FUNCTION_BLOCK FB_TCP_IP
VAR_INPUT
	sName				: STRING := 'SR1000';			(* A kódolvasó neve *)
	sRemoteHost			: STRING(15) := '127.0.0.1';	(* IP adress of remote server *)
	nRemotePort			: UDINT := 9004;				(* SR1000 default port *)
END_VAR
VAR_OUTPUT
END_VAR
VAR
	fbConnect 			:FB_SocketConnect;
	fbSend 				:FB_SocketSend;
	fbReceive 			:FB_SocketReceive;
	fbClose				:FB_SocketClose;
	sTxBuffer			:STRING;
	sRxBuffer			:STRING;
	nStep				:INT := 0;
	
	_ConnectTimeout		:TIME;
	_SendTimeout		:TIME;
	_ReceiveTimeout		:TIME;
	_CloseTimeout		:TIME;

END_VAR

(*
fbConnect(
	sSrvNetId:= '', 
	sRemoteHost:= sRemoteHost, 
	nRemotePort:= nRemotePort, 
	bExecute:= , 
	tTimeout:= _ConnectTimeout, 
	bBusy=> , 
	bError=> , 
	nErrId=> , 
	hSocket=> );
	
fbSend(
	sSrvNetId:= '', 
	hSocket:= fbConnect.hSocket, 
	cbLen:= INT_TO_UDINT(LEN(sTxBuffer)), 
	pSrc:= ADR(sTxBuffer), 
	bExecute:= , 
	tTimeout:= _SendTimeout, 
	bBusy=> , 
	bError=> , 
	nErrId=> );

fbReceive(
	sSrvNetId:= '', 
	hSocket:= fbConnect.hSocket, 
	cbLen:= SIZEOF(sRxBuffer), 
	pDest:= ADR(sRxBuffer), 
	bExecute:= , 
	tTimeout:= _ReceiveTimeout, 
	bBusy=> , 
	bError=> , 
	nErrId=> , 
	nRecBytes=> );

fbClose(
	sSrvNetId:= '', 
	hSocket:= fbConnect.hSocket, 
	bExecute:= , 
	tTimeout:= , 
	bBusy=> , 
	bError=> , 
	nErrId=> );	
	
*)

PROPERTY p_CloseTimeout :  TIME
GET
p_CloseTimeout := _CloseTimeout;
END_GET
SET
IF p_CloseTimeout > T#100MS AND p_CloseTimeout <  T#60S THEN
	_CloseTimeout := p_CloseTimeout;
ELSE
	_CloseTimeout := T#1S;					// default value
END_IF
END_SET
END_PROPERTY

PROPERTY p_ConnectTimeout : TIME
GET
p_ConnectTimeout := _ConnectTimeout;
END_GET
SET
IF p_ConnectTimeout > T#100MS AND p_ConnectTimeout <  T#60S THEN
	_ConnectTimeout := p_ConnectTimeout;
ELSE
	_ConnectTimeout := T#1S;					// default value
END_IF
END_SET
END_PROPERTY

PROPERTY p_ReceiveTimeout : TIME
GET
p_ReceiveTimeout := _ReceiveTimeout;
END_GET
SET
IF p_ReceiveTimeout > T#100MS AND p_ReceiveTimeout <  T#60S THEN
	_ReceiveTimeout := p_ReceiveTimeout;
ELSE
	_ReceiveTimeout := T#1S;					// default value
END_IF
END_SET
END_PROPERTY

PROPERTY p_SendTimeout : TIME
GET
p_SendTimeout := _SendTimeout;
END_GET
SET
IF p_SendTimeout > T#100MS AND p_SendTimeout <  T#60S THEN
	_SendTimeout := p_SendTimeout;
ELSE
	_SendTimeout := T#1S;					// default value
END_IF
END_SET
END_PROPERTY

METHOD ReadSR1000 : BOOL
VAR_INPUT
	sCode						:REFERENCE TO STRING;
	nErrorId					:REFERENCE TO UDINT;
END_VAR
TCP_Com();
ReadSR1000 := FALSE;
CASE nStep OF
0:		fbConnect.bExecute := TRUE;
		sRxBuffer := '';
		nStep := nStep + 20;
	
20:		IF NOT fbConnect.bBusy THEN
			fbConnect.bExecute := FALSE;
			nStep := nStep + 20;
		ELSIF fbConnect.bError THEN
			sCode := '';
			nErrorId := fbConnect.nErrId;
			fbConnect.bExecute := FALSE;
			nStep := 200;
		END_IF
	
40:		sTxBuffer := 'LON$R$N';
		fbSend.bExecute := TRUE;
		nStep := nStep + 20;
	
60:		IF NOT fbSend.bBusy THEN
			fbSend.bExecute := FALSE;
			nStep := 100;
		ELSIF fbSend.bError THEN
			sCode := '';
			nErrorId := fbSend.nErrId;
			fbSend.bExecute := FALSE;
			nStep := 200;
		END_IF
	
100:	fbReceive.bExecute := TRUE;
		nStep := nStep + 20;
	
120:	IF NOT fbReceive.bBusy THEN
			IF NOT fbReceive.bError THEN
					fbReceive.bExecute := FALSE;
					nStep := nStep + 20;
			ELSE
					sCode := '';
					nErrorId := fbReceive.nErrId;
					fbReceive.bExecute := FALSE;
					nStep := 200;
			END_IF
		END_IF

140:	IF fbReceive.nRecBytes > 0 THEN
				IF MID(sRxBuffer, 1, UDINT_TO_INT(fbReceive.nRecBytes)) = '$0D' THEN
					nErrorId := fbReceive.nErrId;
					sCode := LEFT(sRxBuffer, UDINT_TO_INT(fbReceive.nRecBytes)-1);
					nStep := 200;
				ELSE				
					nStep := 100;
				END_IF
		ELSE
				nStep := 100;
		END_IF
		
200:	fbClose.bExecute := TRUE;
		nStep := nStep + 20;
	
220:	IF NOT fbClose.bBusy THEN
			fbClose.bExecute := FALSE;
			nStep := 500;
		ELSIF fbClose.bError THEN
			sCode := '';
			nErrorId := fbClose.nErrId;
			fbClose.bExecute := FALSE;
			nStep := 500;
		END_IF

500:
		ReadSR1000 := TRUE;
		nStep := 0;
END_CASE
END_METHOD

METHOD PRIVATE TCP_Com : BOOL
VAR_INPUT
END_VAR
fbConnect(
	sSrvNetId:= '', 
	sRemoteHost:= sRemoteHost, 
	nRemotePort:= nRemotePort, 
	bExecute:= , 
	tTimeout:= _ConnectTimeout, 
	bBusy=> , 
	bError=> , 
	nErrId=> , 
	hSocket=> );
	
fbSend(
	sSrvNetId:= '', 
	hSocket:= fbConnect.hSocket, 
	cbLen:= INT_TO_UDINT(LEN(sTxBuffer)), 
	pSrc:= ADR(sTxBuffer), 
	bExecute:= , 
	tTimeout:= _SendTimeout, 
	bBusy=> , 
	bError=> , 
	nErrId=> );

fbReceive(
	sSrvNetId:= '', 
	hSocket:= fbConnect.hSocket, 
	cbLen:= SIZEOF(sRxBuffer), 
	pDest:= ADR(sRxBuffer), 
	bExecute:= , 
	tTimeout:= _ReceiveTimeout, 
	bBusy=> , 
	bError=> , 
	nErrId=> , 
	nRecBytes=> );

fbClose(
	sSrvNetId:= '', 
	hSocket:= fbConnect.hSocket, 
	bExecute:= , 
	tTimeout:= , 
	bBusy=> , 
	bError=> , 
	nErrId=> );
END_METHOD

END_FUNCTION_BLOCK

(* stored: Version 1.1.0.1, ProductVersion 3.1.4024.6
   POU FB_TCP_IP: Id {c1992312-48d2-4717-b75b-dedc24e610ec}, SpecialFunc None
   Property p_CloseTimeout: Id {33efcc88-4d1f-4a0d-a66f-024f934a305e}
   Get Get: Id {4966c05f-1d94-411b-965b-58a684b4f3ab}
   Set Set: Id {292f1ddb-7331-4589-985f-101eb2259b4c}
   Property p_ConnectTimeout: Id {68ecfdb7-b451-4f54-8bd2-8444a4217bd6}
   Get Get: Id {eb607fda-6909-4f86-92d4-ac9010a2d0cf}
   Set Set: Id {0e6be276-9ba1-473f-b24d-bec570ef9f1a}
   Property p_ReceiveTimeout: Id {6404b7be-21a9-4f82-afde-9c4caf99ac5c}
   Get Get: Id {5f6211ca-a6c7-4229-be2c-432fd78345cb}
   Set Set: Id {2f7f67d5-dfa2-441c-ad3b-be678a1a0e96}
   Property p_SendTimeout: Id {40941df4-96e4-4d20-b218-a904a47fa97c}
   Get Get: Id {8de5fe80-9f61-48cc-9420-8ad10714abdc}
   Set Set: Id {f9fe7f6a-b01b-4c3c-ba2e-87be848c6417}
   Method ReadSR1000: Id {7d109c9e-4119-4422-a584-cc1ea3132383}
   Method TCP_Com: Id {6fb11f8f-d5c4-409d-9054-2d5f0d95f976} *)
